// TIA Portal V19 export
FUNCTION "LAF_ReadCycleLimits" : Void   // FC77, LAD
TITLE = LAF_ReadCycleLimits
AUTHOR : Siemens Digital Industries
FAMILY : LAF
VERSION : 1.2
// This blocks reads and converts the configured maximum and minimum cycle times.
// stored: Access Published, IsIECCheckEnabled true, SetENOAutomatically false
   VAR_OUTPUT
      maxCycleTime : UInt;   // Configured maximum cycle time
      minCycleTime : UInt;   // Configured minimum cycle time
   END_VAR
   VAR_IN_OUT
      maxComLoad : Int;   // Configured maximum communication load
   END_VAR
   VAR_TEMP
      tempStndPrevCycle : LTime;   // Current plc cycle time / Aktuelle CPU Zykluszeit
      tempRetVal1 : Int;   // Ret_Val / Rückgabewert
      tempRetVal2 : Int;   // Ret_Val / Rückgabewert
      tempRetVal3 : Int;   // Ret_Val / Rückgabewert
      tempUlint : ULInt;   // Temp UInt / Temporär UInt
      tempReal : ULInt;   // Temp Real / Temporär Real
   END_VAR
   VAR_TEMP   // added for the SCL form of the ladder/FBD networks
      _w1 : Bool;
   END_VAR
BEGIN

REGION Network 1: BLOCK INFO HEADER
   // SIEMENS AG / (c)Copyright 2024
   // ------------------------------------------------------------------------------
   // Title:            LAF_ReadCycleLimits
   // Comment/Function: This blocks reads and converts the configured maximum and minimum cycle times.
   // Library/Family:   Library of Automation Framework
   // Author:                Siemens Digital Industry
   // Tested with:       S7-PLCSIM Advanced 6.0
   // Engineering:      TIA Portal V19
   // Restrictions:       ---
   // Requirements:   ---
   // ------------------------------------------------------------------------------
   // Change log table:
   // Version  | Date       | Expert in charge       | Changes applied
   // ---------|------------|------------------------|------------------------------
   // 01.01.00 | 21.06.2024 | SIMATIC Systems Support
   //                         First released version
   // 01.02.00 | 30.09.2024 | SIMATIC Systems Support
   //                         Block information properties updated
END_REGION

REGION Network 2: DESCRIPTION
   // This block retrieves and converts the configured maximum and minimum cycle times, as well as the configured maximum communication load of the system. These values are then stored for subsequent use in the application.
END_REGION

REGION Network 3: Read configured max. cycle time / SPS: Hardwarekonfiguration Einstellungen
   // Cycle monitoring time
   // Maximum permitted duration of the CPU program. If the cycle time exceeds the cycle monitoring time, the CPU goes to STOP or calls a time error OB.
   // Auslesen der minimal und maximal erlaubten Zykluszeit der SPS
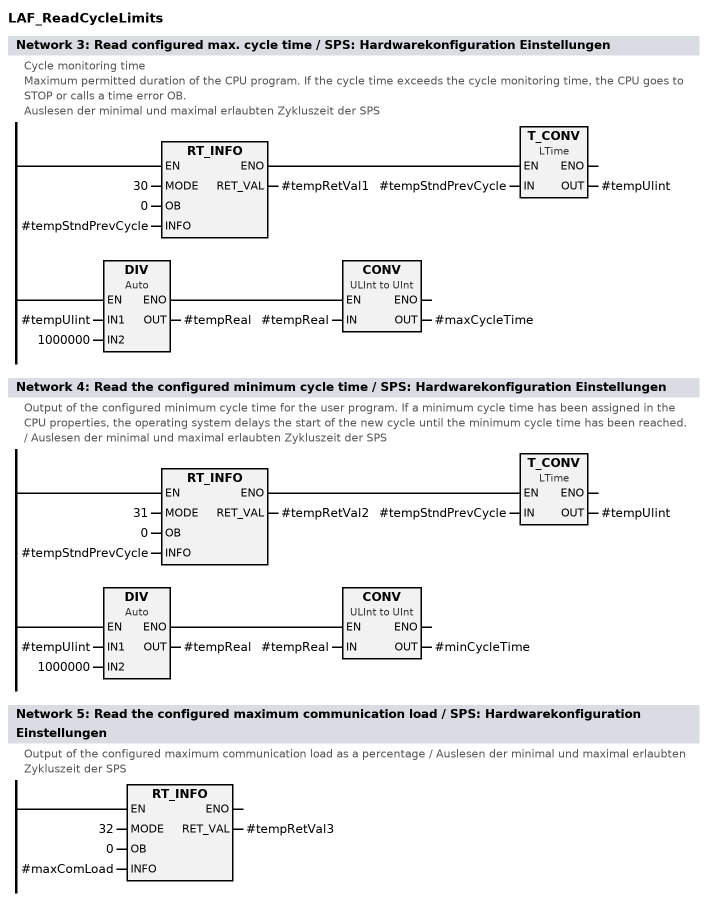
   RUNG wire#powerrail
      RT_INFO(MODE := 30, OB := 0, INFO := #tempStndPrevCycle, Ret_Val => #tempRetVal1)
      { S7_Templates := "[src_type := LTime, dest_type := ULInt]" } T_CONV(IN := #tempStndPrevCycle, OUT => #tempUlint)
   END_RUNG
   RUNG wire#powerrail
      Div(in1 := #tempUlint, in2 := 1000000, out => #tempReal)
      { S7_Templates := "[SrcType := ULInt, DestType := UInt]" } Convert(in := #tempReal, out => #maxCycleTime)
   END_RUNG
   // the same network as SCL:
   #tempRetVal1 := RT_INFO(MODE := 30, OB := 0, INFO := #tempStndPrevCycle, ENO => #_w1);
   IF #_w1 THEN T_CONV(IN := #tempStndPrevCycle, OUT => #tempUlint); END_IF;
   #tempReal := #tempUlint / 1000000;
   #maxCycleTime := ULINT_TO_UINT(#tempReal);
END_REGION

REGION Network 4: Read the configured minimum cycle time / SPS: Hardwarekonfiguration Einstellungen
   // Output of the configured minimum cycle time for the user program. If a minimum cycle time has been assigned in the CPU properties, the operating system delays the start of the new cycle until the minimum cycle time has been reached. / Auslesen der minimal und maximal erlaubten Zykluszeit der SPS
   RUNG wire#powerrail
      RT_INFO(MODE := 31, OB := 0, INFO := #tempStndPrevCycle, Ret_Val => #tempRetVal2)
      { S7_Templates := "[src_type := LTime, dest_type := ULInt]" } T_CONV(IN := #tempStndPrevCycle, OUT => #tempUlint)
   END_RUNG
   RUNG wire#powerrail
      Div(in1 := #tempUlint, in2 := 1000000, out => #tempReal)
      { S7_Templates := "[SrcType := ULInt, DestType := UInt]" } Convert(in := #tempReal, out => #minCycleTime)
   END_RUNG
   // the same network as SCL:
   #tempRetVal2 := RT_INFO(MODE := 31, OB := 0, INFO := #tempStndPrevCycle, ENO => #_w1);
   IF #_w1 THEN T_CONV(IN := #tempStndPrevCycle, OUT => #tempUlint); END_IF;
   #tempReal := #tempUlint / 1000000;
   #minCycleTime := ULINT_TO_UINT(#tempReal);
END_REGION

REGION Network 5: Read the configured maximum communication load / SPS: Hardwarekonfiguration Einstellungen
   // Output of the configured maximum communication load as a percentage / Auslesen der minimal und maximal erlaubten Zykluszeit der SPS
   RUNG wire#powerrail
      RT_INFO(MODE := 32, OB := 0, INFO := #maxComLoad, Ret_Val => #tempRetVal3)
   END_RUNG
   // the same network as SCL:
   #tempRetVal3 := RT_INFO(MODE := 32, OB := 0, INFO := #maxComLoad);
END_REGION
END_FUNCTION
